{attribute 'GeneratedUsingTerminal: EL3413-0000-0016'}
{attribute addProperty BoxType "EL3413-0000-0016"}
{attribute addProperty Id "PM_Inputs_Channel_1AT %I*PM_Inputs_Channel_345EAE5425PM_Inputs_Channel_2AT %I*PM_Inputs_Channel_345EAE5425PM_Inputs_Channel_3AT %I*PM_Inputs_Channel_345EAE5425PM_Inputs_AuxiliaryAT %I*PM_Inputs_Auxiliary_392D510B7PM_Outputs_Channel_1AT %Q*PM_Outputs_Channel_E5FBDE301PM_Outputs_Channel_2AT %Q*PM_Outputs_Channel_E5FBDE301PM_Outputs_Channel_3AT %Q*PM_Outputs_Channel_E5FBDE301PM_Outputs_AuxiliaryAT %Q*PM_Outputs_Auxiliary_6BC1946F2WcStateAT %I*WcState_9091E0EB2InfoDataAT %I*InfoData_32EB74EA10"}
{attribute addProperty CRC "90429588"}
{attribute addProperty Size "99"}
TYPE EL3413_0563D894 EXTENDS EtcSlaveTerminalBase_947E5A46 :
STRUCT
	{attribute addProperty Name "PM_Inputs_Channel_1"}
	PM_Inputs_Channel_1 : PM_Inputs_Channel_345EAE54;
	{attribute addProperty Name "PM_Inputs_Channel_2"}
	PM_Inputs_Channel_2 : PM_Inputs_Channel_345EAE54;
	{attribute addProperty Name "PM_Inputs_Channel_3"}
	PM_Inputs_Channel_3 : PM_Inputs_Channel_345EAE54;
	{attribute addProperty Name "PM_Inputs_Auxiliary"}
	PM_Inputs_Auxiliary : PM_Inputs_Auxiliary_392D510B;
	{attribute addProperty Name "PM_Outputs_Channel_1"}
	PM_Outputs_Channel_1 : PM_Outputs_Channel_E5FBDE30;
	{attribute addProperty Name "PM_Outputs_Channel_2"}
	PM_Outputs_Channel_2 : PM_Outputs_Channel_E5FBDE30;
	{attribute addProperty Name "PM_Outputs_Channel_3"}
	PM_Outputs_Channel_3 : PM_Outputs_Channel_E5FBDE30;
	{attribute addProperty Name "PM_Outputs_Auxiliary"}
	PM_Outputs_Auxiliary : PM_Outputs_Auxiliary_6BC1946F;
	{attribute addProperty Name "WcState"}
	WcState : WcState_9091E0EB;
	{attribute addProperty Name "InfoData"}
	InfoData : InfoData_32EB74EA;
END_STRUCT
END_TYPE

(* stored: Version 1.2.0.0, ProductVersion 3.1.4024.9
   DUT EL3413_0563D894: Id {75eb92e9-ec3f-4db6-b3ff-9a1955d5a606} *)
